Staubli VAL3: removeString.pgx

public program removeString(string& x_sInput[], num x_nStart, num x_nEnd, string& x_sResult[])
  local num l_nElement
  local num l_nLength
  local string l_sLeft
  local string l_sRigt
  local string l_sRight
begin

  l_nLength = size(x_sInput)
  resize(x_sResult,1,1)
  x_sResult =""
  resize(x_sResult,1,l_nLength)

  // iterate complete input x_sInput[0] ... x_sInput[l_nLength-1]
  for l_nElement = 0 to l_nLength-1

    // ab cd efghj
    // 12 34 56789 len
    // 01 23 45678 idx
    l_sLeft = left(x_sInput[l_nElement], sel(x_nStart==0, 0, x_nStart))
    l_sRight = right(x_sInput[l_nElement], sel(len(x_sInput[l_nElement])-x_nEnd-1<0, 0, len(x_sInput[l_nElement])-x_nEnd-1))
    x_sResult[l_nElement] = l_sLeft + l_sRight

  endFor


end
